(* CoDeSys 2.3.9.35 project: maquina_de_lava.pro *)
(* Author: Altus *)
(* Libraries: DU35x.lib 7.7.11 15:59:13, Navigation.lib 15.7.11 10:06:00, SysLibTargetVisu.lib 26.11.08 09:53:28, Standard.lib 26.11.08 09:46:20, Iecsfc.lib 26.11.08 09:46:14, SYSLIBCALLBACK.LIB 26.11.08 09:53:30 *)

(* PLC configuration (modules and I/O channels)
Comunicação [Comunica] node 0, in %IB0 out %QB0
  COM1 [COM1] node 0, in %IB0 out %QB0 {BaudRate = 115200; Paridade = Sem Paridade; StopBits = 1 Stop Bit; Modem = Sem RTS/CTS; Delay = 5}
    MToolIEC [Codesys] node 0, in %IB0 out %QB0
  COM2 [COM2] node 1, in %IB0 out %QB0 {BaudRate = 115200; Paridade = Sem Paridade; StopBits = 1 Stop Bit; Modem = Sem RTS/CTS; Delay = 5}
    Desabilitada [Desabilitado485] node 0, in %IB0 out %QB0
Entradas Digitais 0 [Entradas0] node 0, in %IW0 out %QB0
  I00 AT %IX0.0 [BitInput] I0.0
  I01 AT %IX0.1 [BitInput] I0.1
  I02 AT %IX0.2 [BitInput] I0.2
  I03 AT %IX0.3 [BitInput] I0.3
  I04 AT %IX0.4 [BitInput] I0.4
  I05 AT %IX0.5 [BitInput] I0.5
  I06 AT %IX0.6 [BitInput] I0.6
  I07 AT %IX0.7 [BitInput] I0.7
  I08 AT %IX0.8 [BitInput] I0.8
Entradas Digitais 1 [Entradas1] node 0, in %IW1 out %QB0
  I10 AT %IX1.0 [BitInput] I1.0
  I11 AT %IX1.1 [BitInput] I1.1
  I12 AT %IX1.2 [BitInput] I1.2
  I13 AT %IX1.3 [BitInput] I1.3
  I14 AT %IX1.4 [BitInput] I1.4
  I15 AT %IX1.5 [BitInput] I1.5
  I16 AT %IX1.6 [BitInput] I1.6
  I17 AT %IX1.7 [BitInput] I1.7
  I18 AT %IX1.8 [BitInput] I1.8
Entradas Digitais 2 [Entradas2] node 0, in %IW2 out %QB0
  I20 AT %IX2.0 [BitInput] I2.0
  I21 AT %IX2.1 [BitInput] I2.1
AI0 AT %IW4 [WordInput] AI0 {TipoAnalogica = Tensão 0-10V; FiltroAnalogica = Filtro 0 - AI=2ms  / AV=90ms; FundoEscala = 10}
AI1 AT %IW5 [WordInput] AI1 {TipoAnalogica = Channel Disable; FiltroAnalogica = Filter 0 - AI=2ms  / AV=90ms; FundoEscala = 0}
AI2 AT %IW6 [WordInput] AI2 {TipoAnalogica = Channel Disable; FiltroAnalogica = Filter 0 - AI=2ms  / AV=90ms; FundoEscala = 0}
AI3 AT %IW7 [WordInput] AI3 {TipoAnalogica = Channel Disable; FiltroAnalogica = Filter 0 - AI=2ms  / AV=90ms; FundoEscala = 0}
Bloco 0 [Bloco0] node 0, in %IB16 out %QB0
  Desabilitado [DesabilitadoBloco0] node 0, in %IB16 out %QB0
Bidirecional [BidirecionalBloco1] node 0, in %IB16 out %QB0 {ContagemBidirecional = Quadratura 2x}
Contador 0 [EntradaConfContador0] node 0, in %IB16 out %QB0 {EntradaConfiguravelContador = Desabilitada}
Contador 2 [EntradaConfContador2] node 0, in %IB16 out %QB0 {EntradaConfiguravelContador = Zeramento}
Saídas Digitais 0 [Saidas0] node 0, in %IW0 out %QW0
  Q00 AT %QX0.0 [BitOutput] Q0.0
  Q01 AT %QX0.1 [BitOutput] Q0.1
  Q02 AT %QX0.2 [BitOutput] Q0.2
  Q03 AT %QX0.3 [BitOutput] Q0.3
  Q04 AT %QX0.4 [BitOutput] Q0.4
  Q05 AT %QX0.5 [BitOutput] Q0.5
  Q06 AT %QX0.6 [BitOutput] Q0.6
  Q07 AT %QX0.7 [BitOutput] Q0.7
Saídas Digitais 1 [Saidas1] node 0, in %IW0 out %QW1
  Q10 AT %QX1.0 [BitOutput] Q1.0
  Q11 AT %QX1.1 [BitOutput] Q1.1
  Q12 AT %QX1.2 [BitOutput] Q1.2
  Q13 AT %QX1.3 [BitOutput] Q1.3
  Q14 AT %QX1.4 [BitOutput] Q1.4
  Q15 AT %QX1.5 [BitOutput] Q1.5
  Q16 AT %QX1.6 [BitOutput] Q1.6
  Q17 AT %QX1.7 [BitOutput] Q1.7
AO0 AT %QW3 [WordOutput] AO0 {TipoAnalogica = Channel Disable; FundoEscala = 0}
AO1 AT %QW4 [WordOutput] AO1 {TipoAnalogica = Tensão 0-10V; FundoEscala = 10}
Saída Rápida 0 Desabilitada [DesabilitadoF0] node 0, in %IB0 out %QB10
PTO [PTOF1] node 1, in %IB0 out %QB10 {RampaPTO = Trapezoidal}
Saídas Comum de Contador [SaidasContador] node 2, in %IB0 out %QB10
  Saída do Bloco 0 Desabilitada [DesabilitadoSaidaBloco0] node 0, in %IB0 out %QB10
  Saída do Bloco 1 Desabilitada [DesabilitadoSaidaBloco1] node 1, in %IB0 out %QB10
Eventos Externos [Eventos] node 2, in %IB13 out %QB6
  Evento Temporizado [TimerEvent] node 0, in %IB13 out %QB6 {Intervalo = 10}
*)

(* Task configuration *)
TASK PRINCIPAL (PRIORITY := 1, INTERVAL := T#1ms);
	PLC_PRG();
END_TASK
TASK NAVIGATION (PRIORITY := 1, INTERVAL := T#20ms);
	NAVEGA();
END_TASK
TASK VISUALIZATION (PRIORITY := 1, INTERVAL := T#500ms);
	MAINTARGETVISU_PAINT_CODE
END_TASK
TASK KEYBOARD_USAGE (PRIORITY := 1, INTERVAL := T#20ms);
	NAVEGA();
END_TASK

(* POU PLC_PRG, LD *)
PROGRAM PLC_PRG
VAR_INPUT
	DESLIGAR 	AT %IX0.1: 	BOOL;
	LIGAR		AT %IX0.0: 	BOOL;
	MN 			AT %IX0.2: 	BOOL;
	MR 			AT %IX0.3: 	BOOL;
	MT 			AT %IX0.4: 	BOOL;
	POT 		AT %IW4: 	WORD;	(*ENTRADA DA LEITURA DO POTENCIOMENTRO*)
END_VAR

VAR_OUTPUT
	SENT_ROTA 	AT %QX0.2: 	BOOL;	(*SENTIDO DE ROTACAO DO MOTOR 0= HORARIO 1= ANT-HORARIO*)
	HAB_MOTOR 	AT %QX0.3: 	BOOL;	(*HABILITA O MOTOR 1=BONINAS PERMANECE ENERGIZADAS 0=BONINAS ENERGIZADAS PENAS DURANTE O MOVIMENTO*)
	PLS_QTD 	AT %QX0.4: 	BOOL;	(*QUANTIDADE DE PULSOS 0= 200 PULOS PARA UMA VOLTA 1=400 PULOS PARA UMA VOLTA*)
	ZERAR 		AT %QX0.0: 	BOOL;	(*SAIDA UTILIZADO PARA ZERAR O CONTADOR*)
END_VAR

VAR
	FREQ 		AT %MD1652: 	DWORD;	(*FREQUENCIA DO SINA DE SAIDA*)
	PLS_TOT 	AT %MD1653: 	DWORD;	(*NUMERO DE PULSOS TOTAL*)
	PLS_RAMP 	AT %MD1654: 	DWORD; 	(*NUMERO DE PULSOS POR RAMPA DE ACELARACAO/DESACELERACAO*)
	START_MOTOR AT %MX3314.2: 	BOOL; 	(*ACIONAR O DISPARO DOS PULSOS NA SAIDA RAPAIDA*)
	STOP_MOTOR 	AT %MX3314.3: 	BOOL; 	(*PARA O DISPARO DOS PULSOS NA SAIDA RAPAIDA*)
	CONTADOR 	AT %MD1633:		DWORD;	(*ENTRADA RAPIDA PARA ACESSAR O CONTADOR 2 LIGADO AO ENCODER*)
	PARAR 		AT %MX3276.1: 	BOOL;	(*PARAR O CONTADOR*)
	PLS_CONT: 		REAL; 				(*NUMERO DE PULSOS CONTADOS*)
	AUX_PLS_CONT: 	DWORD;
	ROTACAO: 		REAL	:=0;
	RPM: 			REAL	:=0;
	AUX_RPM: 		REAL;
	SMN: 			BOOL;
	SMR: 			BOOL;
	SMT: 			BOOL;
	LIGADO: 		BOOL;
	AUX_POT: 		REAL;
	AUX_POT0: 		REAL;
	AUX_POT1: 		REAL;
	AUX_POT2: 		REAL;
	AUX_POT11: 		DWORD;
	AUX_POT22:		DWORD;
	ADD1: 			REAL;
	ADD2:			REAL;
	ADD3: 			REAL;
	AUX1: 			BOOL;
	AUX_READ: 		BOOL;
	TEMP_RH: 		TON;
	TEMP_RAH: 		TOF;
	TEMP_READ: 		TON;
	TEMP_DELAY: 	TON;
	AUX_TIME: 		INT 	:= 2000;
	FINAL_TIME: 	TIME;
	MULT: 			REAL;
	FREQ1: 			DWORD;
	FREQ2: 			DWORD;
	FREQ3: 			DWORD;
END_VAR
VAR (* helpers for the ST form of the networks *)
	_p1 : BOOL;
	_p2 : BOOL;
END_VAR
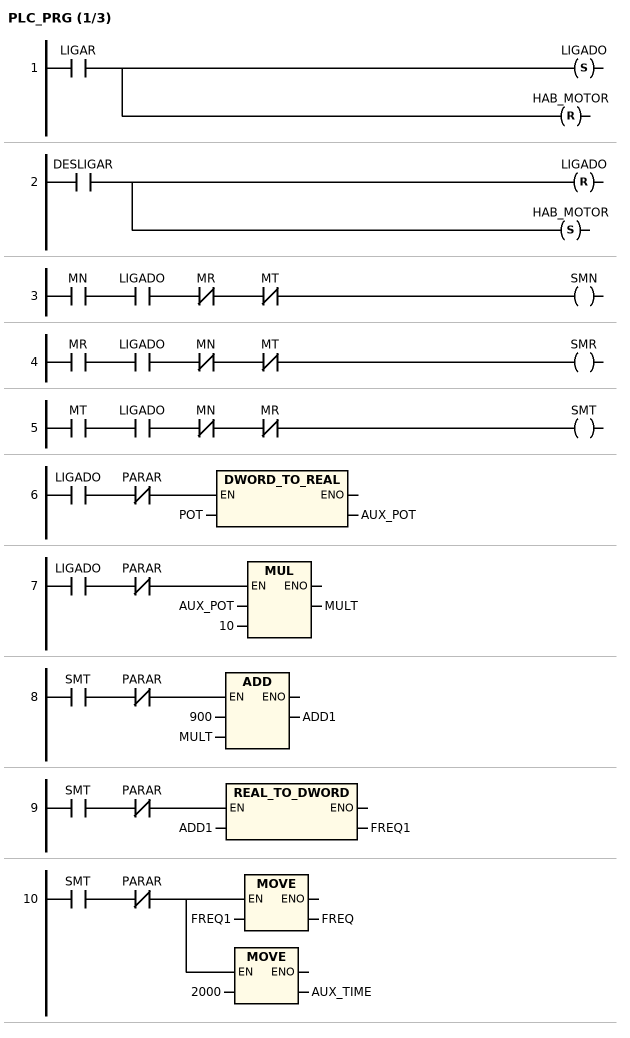
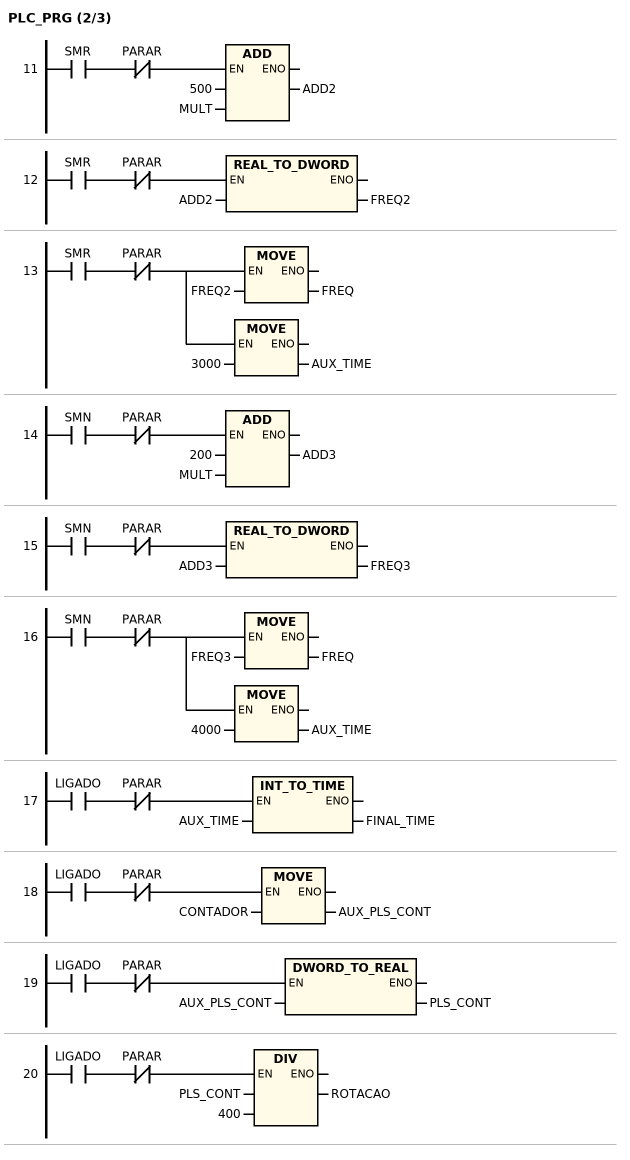
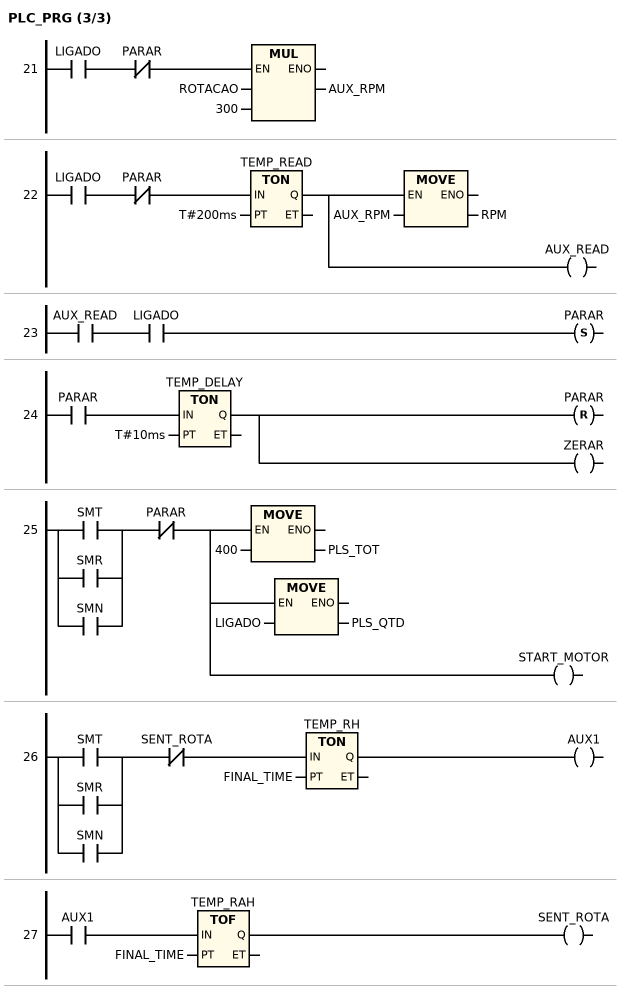
_LD_ (* Ladder Diagram *)
NETWORK 1
	[LIGAR] --- (S LIGADO) (R HAB_MOTOR)
NETWORK 2
	[DESLIGAR] --- (R LIGADO) (S HAB_MOTOR)
NETWORK 3
	[MN] - [LIGADO] - [/MR] - [/MT] --- (SMN)
NETWORK 4
	[MR] - [LIGADO] - [/MN] - [/MT] --- (SMR)
NETWORK 5
	[MT] - [LIGADO] - [/MN] - [/MR] --- (SMT)
NETWORK 6
	[LIGADO] - [/PARAR]
		EN --- DWORD_TO_REAL(POT) => AUX_POT
NETWORK 7
	[LIGADO] - [/PARAR]
		EN --- MUL(AUX_POT, 10) => MULT
NETWORK 8
	[SMT] - [/PARAR]
		EN --- ADD(900, MULT) => ADD1
NETWORK 9
	[SMT] - [/PARAR]
		EN --- REAL_TO_DWORD(ADD1) => FREQ1
NETWORK 10
	[SMT] - [/PARAR]
		EN --- MOVE(FREQ1) => FREQ
		EN --- MOVE(2000) => AUX_TIME
NETWORK 11
	[SMR] - [/PARAR]
		EN --- ADD(500, MULT) => ADD2
NETWORK 12
	[SMR] - [/PARAR]
		EN --- REAL_TO_DWORD(ADD2) => FREQ2
NETWORK 13
	[SMR] - [/PARAR]
		EN --- MOVE(FREQ2) => FREQ
		EN --- MOVE(3000) => AUX_TIME
NETWORK 14
	[SMN] - [/PARAR]
		EN --- ADD(200, MULT) => ADD3
NETWORK 15
	[SMN] - [/PARAR]
		EN --- REAL_TO_DWORD(ADD3) => FREQ3
NETWORK 16
	[SMN] - [/PARAR]
		EN --- MOVE(FREQ3) => FREQ
		EN --- MOVE(4000) => AUX_TIME
NETWORK 17
	[LIGADO] - [/PARAR]
		EN --- INT_TO_TIME(AUX_TIME) => FINAL_TIME
NETWORK 18
	[LIGADO] - [/PARAR]
		EN --- MOVE(CONTADOR) => AUX_PLS_CONT
NETWORK 19
	[LIGADO] - [/PARAR]
		EN --- DWORD_TO_REAL(AUX_PLS_CONT) => PLS_CONT
NETWORK 20
	[LIGADO] - [/PARAR]
		EN --- DIV(PLS_CONT, 400) => ROTACAO
NETWORK 21
	[LIGADO] - [/PARAR]
		EN --- MUL(ROTACAO, 300) => AUX_RPM
NETWORK 22
	[LIGADO] - [/PARAR] - TEMP_READ:TON(IN: *, PT: T#200ms) --- (AUX_READ)
		EN --- MOVE(AUX_RPM) => RPM
NETWORK 23
	[AUX_READ] - [LIGADO] --- (S PARAR)
NETWORK 24
	[PARAR] - TEMP_DELAY:TON(IN: *, PT: T#10ms) --- (R PARAR) (ZERAR)
NETWORK 25
	{ [SMT] | [SMR] | [SMN] } - [/PARAR] --- (START_MOTOR)
		EN --- MOVE(400) => PLS_TOT
		EN --- MOVE(LIGADO) => PLS_QTD
NETWORK 26
	{ [SMT] | [SMR] | [SMN] } - [/SENT_ROTA] - TEMP_RH:TON(IN: *, PT: FINAL_TIME) --- (AUX1)
NETWORK 27
	[AUX1] - TEMP_RAH:TOF(IN: *, PT: FINAL_TIME) --- (SENT_ROTA)
_END_LD_
(* the same logic as Structured Text *)
(* Network 1 *)
IF LIGAR THEN LIGADO := TRUE; HAB_MOTOR := FALSE; END_IF;
(* Network 2 *)
IF DESLIGAR THEN LIGADO := FALSE; HAB_MOTOR := TRUE; END_IF;
(* Network 3 *)
SMN := MN AND LIGADO AND NOT MR AND NOT MT;
(* Network 4 *)
SMR := MR AND LIGADO AND NOT MN AND NOT MT;
(* Network 5 *)
SMT := MT AND LIGADO AND NOT MN AND NOT MR;
(* Network 6 *)
IF LIGADO AND NOT PARAR THEN
	AUX_POT := DWORD_TO_REAL(POT);
END_IF;
(* Network 7 *)
IF LIGADO AND NOT PARAR THEN
	MULT := AUX_POT * 10;
END_IF;
(* Network 8 *)
IF SMT AND NOT PARAR THEN
	ADD1 := 900 + MULT;
END_IF;
(* Network 9 *)
IF SMT AND NOT PARAR THEN
	FREQ1 := REAL_TO_DWORD(ADD1);
END_IF;
(* Network 10 *)
IF SMT AND NOT PARAR THEN
	FREQ := FREQ1;
	AUX_TIME := 2000;
END_IF;
(* Network 11 *)
IF SMR AND NOT PARAR THEN
	ADD2 := 500 + MULT;
END_IF;
(* Network 12 *)
IF SMR AND NOT PARAR THEN
	FREQ2 := REAL_TO_DWORD(ADD2);
END_IF;
(* Network 13 *)
IF SMR AND NOT PARAR THEN
	FREQ := FREQ2;
	AUX_TIME := 3000;
END_IF;
(* Network 14 *)
IF SMN AND NOT PARAR THEN
	ADD3 := 200 + MULT;
END_IF;
(* Network 15 *)
IF SMN AND NOT PARAR THEN
	FREQ3 := REAL_TO_DWORD(ADD3);
END_IF;
(* Network 16 *)
IF SMN AND NOT PARAR THEN
	FREQ := FREQ3;
	AUX_TIME := 4000;
END_IF;
(* Network 17 *)
IF LIGADO AND NOT PARAR THEN
	FINAL_TIME := INT_TO_TIME(AUX_TIME);
END_IF;
(* Network 18 *)
IF LIGADO AND NOT PARAR THEN
	AUX_PLS_CONT := CONTADOR;
END_IF;
(* Network 19 *)
IF LIGADO AND NOT PARAR THEN
	PLS_CONT := DWORD_TO_REAL(AUX_PLS_CONT);
END_IF;
(* Network 20 *)
IF LIGADO AND NOT PARAR THEN
	ROTACAO := PLS_CONT / 400;
END_IF;
(* Network 21 *)
IF LIGADO AND NOT PARAR THEN
	AUX_RPM := ROTACAO * 300;
END_IF;
(* Network 22 *)
TEMP_READ(IN := LIGADO AND NOT PARAR, PT := T#200ms);
_p1 := TEMP_READ.Q;
IF _p1 THEN
	RPM := AUX_RPM;
END_IF;
AUX_READ := _p1;
(* Network 23 *)
IF AUX_READ AND LIGADO THEN PARAR := TRUE; END_IF;
(* Network 24 *)
TEMP_DELAY(IN := PARAR, PT := T#10ms);
IF TEMP_DELAY.Q THEN PARAR := FALSE; END_IF;
ZERAR := TEMP_DELAY.Q;
(* Network 25 *)
_p2 := (SMT OR SMR OR SMN) AND NOT PARAR;
IF _p2 THEN
	PLS_TOT := 400;
	PLS_QTD := LIGADO;
END_IF;
START_MOTOR := _p2;
(* Network 26 *)
TEMP_RH(IN := (SMT OR SMR OR SMN) AND NOT SENT_ROTA, PT := FINAL_TIME);
AUX1 := TEMP_RH.Q;
(* Network 27 *)
TEMP_RAH(IN := AUX1, PT := FINAL_TIME);
SENT_ROTA := TEMP_RAH.Q;
END_PROGRAM

(* POU NAVEGA, ST *)
PROGRAM NAVEGA
VAR
	ControleTelas : NAVIGATION;
	ListaTelas 	: ARRAY [0..30] OF STRING(10);
END_VAR
(* Adiciona a tela MAIN como tela principal *)
ListaTelas[0] := 'MAIN';

(* Ativa o controle automático de navegação somente pelo teclado *)
ControleTelas(ENABLE_UPDW := FALSE, VISU_LIST := ListaTelas, UP := FALSE , DOWN := FALSE);
END_PROGRAM

(* Visualisation MAIN
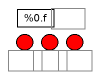
rounded rectangle at (32,3)-(69,21): text "%0.f"; shows PLC_PRG.RPM
ellipse at (31,28)-(48,44): alarm colour if PLC_PRG.SMN
ellipse at (56,28)-(73,44): alarm colour if PLC_PRG.SMR
ellipse at (81,28)-(98,44): alarm colour if PLC_PRG.SMT
4 more shapes without text or variables
*)
